// TIA Portal V18 export
TYPE "MaterialGateUDT"
   STRUCT
      CMD : Struct
         RequestPB : Bool;   // 物料门请求按钮
         RequestPB_Auto : Bool;   // 物料门请求按钮-自动
      END_STRUCT;
      Status : Struct
         "Lock/Unlock Indicator" : Bool;   // 物料门锁定输出状态指示
         "INT" : Int;   // 物料门状态:1:已锁定,2:已解锁,3:安全门被打开
         Locked : Bool;   // 物料门已锁定
         Unlocked : Bool;   // 物料门已解锁
         Opened : Bool;   // 物料门已打开
      END_STRUCT;
   END_STRUCT;
END_TYPE
